FUNCTION_BLOCK FB_mcOperationMode
VAR_INPUT
	eModeRequired : E_mcOperationMode;
END_VAR
VAR_OUTPUT
	eModeActive  : E_mcOperationMode;
END_VAR
VAR
	//	fbMsgAutomaticMode : FB_Messagess;
END_VAR

M_SetMode(eCommand := eModeRequired);

METHOD M_PreCheckAutomatic : BOOL
VAR_INPUT
END_VAR
(*IF Main.fbAxis.Power.Status THEN
	M_PreCheckAutomatic:=TRUE;
//	fbMsgAutomaticMode.Release();
	ELSE
//	fbMsgAutomaticMode.SendMessage(TC_Events.TC_EventOperationModeAutomatic.AxisPower,'');
    M_PreCheckAutomatic:=FALSE;	
END_IF
*);
END_METHOD

METHOD M_SetMode : HRESULT
VAR_INPUT
	eCommand : E_mcOperationMode;
END_VAR
CASE eCommand OF 
	
E_mcOperationMode.Initialization :
	THIS^.eModeActive:=E_mcOperationMode.Initialization;
	M_SetMode:=F_HRESULTSUCCESS(NOERR);

E_mcOperationMode.Service :
	THIS^.eModeActive:=E_mcOperationMode.Service;
	M_SetMode:=F_HRESULTSUCCESS(NOERR);

E_mcOperationMode.Manual:
	THIS^.eModeActive:=E_mcOperationMode.Manual;
	M_SetMode:=F_HRESULTSUCCESS(NOERR);

E_mcOperationMode.Simulation:
	THIS^.eModeActive:=E_mcOperationMode.Simulation;
	M_SetMode:=F_HRESULTSUCCESS(NOERR);

E_mcOperationMode.Automatic:
	IF M_PreCheckAutomatic () THEN
		THIS^.eModeActive:=E_mcOperationMode.Automatic;
		M_SetMode:=F_HRESULTSUCCESS(NOERR);
	ELSE
		THIS^.eModeRequired:=THIS^.eModeActive;
		M_SetMode:=F_HRESULTFAILURE(DEVICE_NOTREADY);
	END_IF	

ELSE
	M_SetMode:=F_HRESULTFAILURE(DEVICE_INVALIDDATA);

END_CASE
END_METHOD

END_FUNCTION_BLOCK

(* stored: Version 1.1.0.1, ProductVersion 3.1.4024.6
   POU FB_mcOperationMode: Id {838fec8e-ff4c-4564-b383-bdc6fa52ca9e}, SpecialFunc None
   Method M_PreCheckAutomatic: Id {a20a50ea-b80e-4275-be7e-d6401d3e6aa2}
   Method M_SetMode: Id {7d980421-3d62-47dc-a953-9928918ddfc3} *)
